// TIA Portal project "Question 5" (V15)

(* hardware
DEVICE "S71500/ET200MP station_1"  S7-1500 station
   slot 0: "Rail_0"  Rack  6ES7 590-1***0-0AA0
   slot 1: "PLC_1"  Unspecific CPU 1500  6ES7 5XX-XXXXX-XXXX  V2.5
*)

// ===== PLC "PLC_1"  Unspecific CPU 1500 =====

VAR_GLOBAL   // PLC tag table "Default tag table"
   "PB" AT %I0.0 : Bool;
   "Tag_1" AT %M0.0 : Bool;
   "Tag_2" AT %M0.2 : Bool;
   "CONVEYOR" AT %Q0.0 : Bool;
   "Tag_3" AT %M0.1 : Bool;
   "LEVEL SENSOR" AT %I0.1 : Bool;
   "VIBRATORY FEEDER" AT %Q0.1 : Bool;
END_VAR

// folder: System blocks/Program resources

DATA_BLOCK "TIMER_VIB_2S"   // DB1
{ S7_Optimized_Access := 'TRUE' }
AUTHOR : Simatic
FAMILY : IEC
NAME : IEC_TMR
VERSION : 1.0
// stored: InstanceOfName IEC_TIMER
"IEC_TIMER"
BEGIN
END_DATA_BLOCK

DATA_BLOCK "TIMER_CONV2S"   // DB2
{ S7_Optimized_Access := 'TRUE' }
AUTHOR : Simatic
FAMILY : IEC
NAME : IEC_TMR
VERSION : 1.0
// stored: InstanceOfName IEC_TIMER
"IEC_TIMER"
BEGIN
END_DATA_BLOCK

// folder: (top level)

ORGANIZATION_BLOCK "Main"   // OB1, LAD, ProgramCycle
TITLE = "Main Program Sweep (Cycle)"
{ S7_Optimized_Access := 'TRUE' }
VERSION : 0.1
   VAR_INPUT
      Initial_Call : Bool;   // Initial call of this OB
      Remanence : Bool;   // =True, if remanent data are available
   END_VAR
BEGIN

REGION Network 1
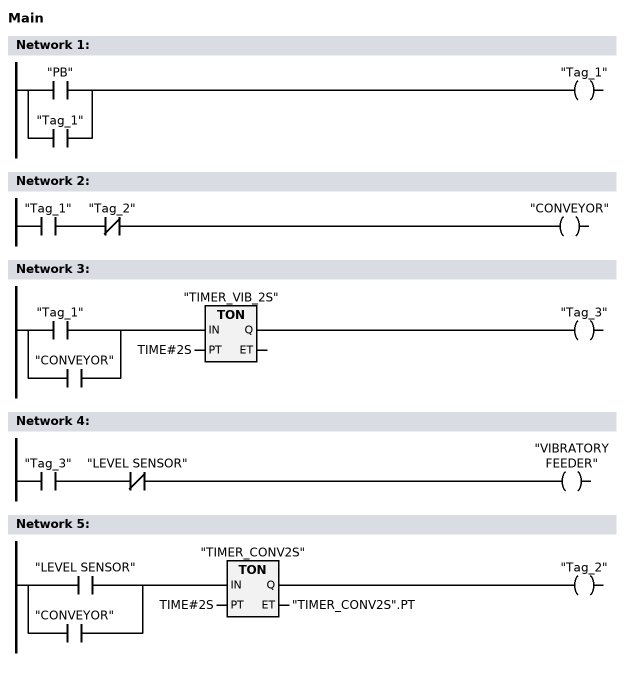
   RUNG wire#powerrail
      Contact( "PB" )
      wire#w1
      Coil( "Tag_1" )
   END_RUNG
   RUNG wire#powerrail
      Contact( "Tag_1" )
   END_RUNG wire#w1
   // the same network as SCL:
   "Tag_1" := "PB" OR "Tag_1";
END_REGION

REGION Network 2
   RUNG wire#powerrail
      Contact( "Tag_1" )
      I_Contact( "Tag_2" )
      Coil( "CONVEYOR" )
   END_RUNG
   // the same network as SCL:
   "CONVEYOR" := "Tag_1" AND NOT "Tag_2";
END_REGION

REGION Network 3
   "TIMER_VIB_2S".TON(IN := "Tag_1" OR "CONVEYOR", PT := TIME#2S);
   "Tag_3" := "TIMER_VIB_2S".Q;
END_REGION

REGION Network 4
   RUNG wire#powerrail
      Contact( "Tag_3" )
      I_Contact( "LEVEL SENSOR" )
      Coil( "VIBRATORY FEEDER" )
   END_RUNG
   // the same network as SCL:
   "VIBRATORY FEEDER" := "Tag_3" AND NOT "LEVEL SENSOR";
END_REGION

REGION Network 5
   "TIMER_CONV2S".TON(IN := "LEVEL SENSOR" OR "CONVEYOR", PT := TIME#2S, ET => "TIMER_CONV2S".PT);
   "Tag_2" := "TIMER_CONV2S".Q;
END_REGION
END_ORGANIZATION_BLOCK